// SIMATIC STEP 7 (V5.x) project PRACTICA PRESELECCIO
// CPU: CPU313 C-2 DP(1)
// station: P_ADR_BUS
// station: Hardware
// station: Equipo SIMATIC 300
// program: Programa S7(1)

SYMBOL_TABLE
"FLANCOS"	DB 1	DB 1
"P PRESELECCION"	I 0.0	BOOL
"EJECUTAR"	I 0.1	BOOL
"P EMERGENCIA"	I 0.2	BOOL
"Cycle Execution"	OB 1	OB 1
"SELECCION BOMBA 1"	Q 0.0	BOOL
"SELECCION BOMBA 2"	Q 0.1	BOOL
"SELECCION BOMBA 3"	Q 0.2	BOOL
"SELECCION BOMBA 4"	Q 0.3	BOOL
"EJECUCION BOMBA 1"	Q 0.4	BOOL
"EJECUCION BOMBA 2"	Q 0.5	BOOL
"EJECUCION BOMBA 3"	Q 0.6	BOOL
"EJECUCION BOMBA 4"	Q 0.7	BOOL
END_SYMBOL_TABLE

DATA_BLOCK "FLANCOS"	// DB 1
VERSION : 0.1
  STRUCT
   M0 : BOOL ;
   M1 : BOOL ;
   M2 : BOOL ;
   M3 : BOOL ;
   M4 : BOOL ;
   M5 : BOOL ;
   M6 : BOOL ;
   M7 : BOOL ;
   M10 : BOOL ;
   M11 : BOOL ;
   M12 : BOOL ;
   M13 : BOOL ;
   M14 : BOOL ;
   M15 : BOOL ;
   M16 : BOOL ;
   M17 : BOOL ;
   M20 : BOOL ;
   M21 : BOOL ;
   M22 : BOOL ;
   M23 : BOOL ;
   M24 : BOOL ;
   M25 : BOOL ;
   M26 : BOOL ;
   M27 : BOOL ;
  END_STRUCT ;	
BEGIN
END_DATA_BLOCK

ORGANIZATION_BLOCK "Cycle Execution"	// OB 1
TITLE = "Main Program Sweep (Cycle)"
VERSION : 0.1
VAR_TEMP
  OB1_EV_CLASS : BYTE ;	//Bits 0-3 = 1 (Coming event), Bits 4-7 = 1 (Event class 1)
  OB1_SCAN_1 : BYTE ;	//1 (Cold restart scan 1 of OB 1), 3 (Scan 2-n of OB 1)
  OB1_PRIORITY : BYTE ;	//Priority of OB Execution
  OB1_OB_NUMBR : BYTE ;	//1 (Organization block 1, OB1)
  OB1_RESERVED_1 : BYTE ;	//Reserved for system
  OB1_RESERVED_2 : BYTE ;	//Reserved for system
  OB1_PREV_CYCLE : INT ;	//Cycle time of previous OB1 scan (milliseconds)
  OB1_MIN_CYCLE : INT ;	//Minimum cycle time of OB1 (milliseconds)
  OB1_MAX_CYCLE : INT ;	//Maximum cycle time of OB1 (milliseconds)
  OB1_DATE_TIME : DATE_AND_TIME ;	//Date and time OB1 started
END_VAR
BEGIN
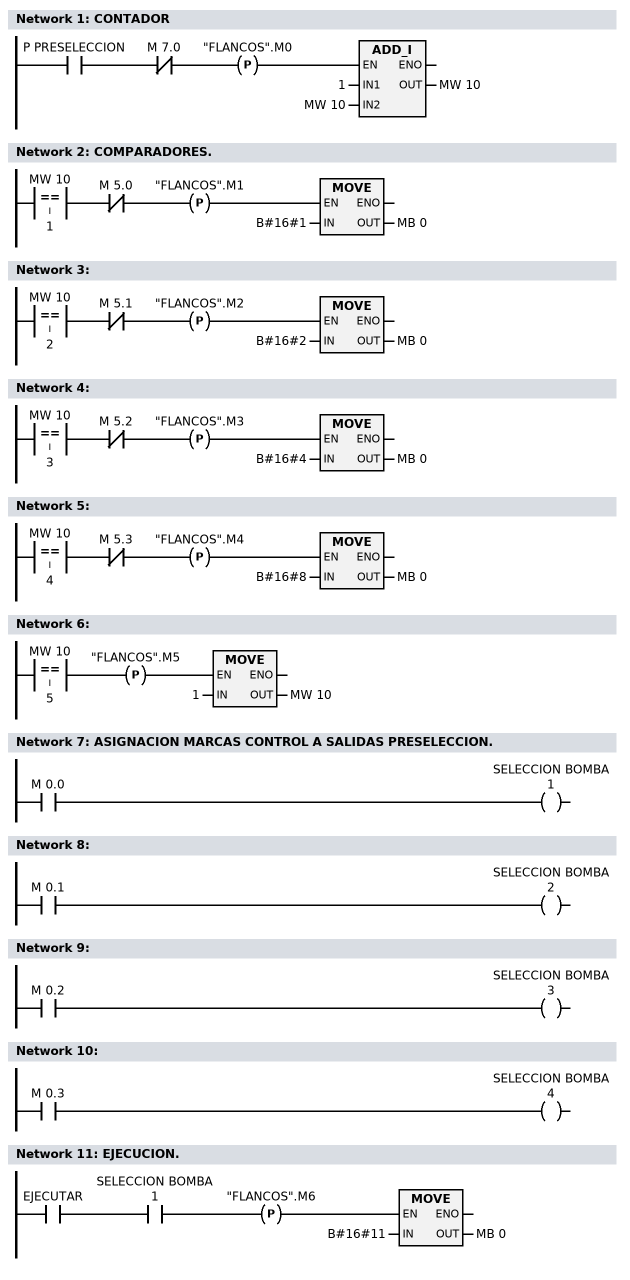
NETWORK
TITLE = CONTADOR
      A     "P PRESELECCION";
      AN    M 7.0;
      FP    "FLANCOS".M0;
      JNB   _001;
      L     1;
      L     MW 10;
      +I;
      T     MW 10;
_001: NOP   0;
NETWORK
TITLE = COMPARADORES.
      A(;
      L     MW 10;
      L     1;
      ==I;
      );
      AN    M 5.0;
      FP    "FLANCOS".M1;
      JNB   _002;
      L     B#16#1;
      T     MB 0;
_002: NOP   0;
NETWORK
TITLE =
      A(;
      L     MW 10;
      L     2;
      ==I;
      );
      AN    M 5.1;
      FP    "FLANCOS".M2;
      JNB   _003;
      L     B#16#2;
      T     MB 0;
_003: NOP   0;
NETWORK
TITLE =
      A(;
      L     MW 10;
      L     3;
      ==I;
      );
      AN    M 5.2;
      FP    "FLANCOS".M3;
      JNB   _004;
      L     B#16#4;
      T     MB 0;
_004: NOP   0;
NETWORK
TITLE =
      A(;
      L     MW 10;
      L     4;
      ==I;
      );
      AN    M 5.3;
      FP    "FLANCOS".M4;
      JNB   _005;
      L     B#16#8;
      T     MB 0;
_005: NOP   0;
NETWORK
TITLE =
      A(;
      L     MW 10;
      L     5;
      ==I;
      );
      FP    "FLANCOS".M5;
      JNB   _006;
      L     1;
      T     MW 10;
_006: NOP   0;
NETWORK
TITLE = ASIGNACION MARCAS CONTROL A SALIDAS PRESELECCION.
      A     M 0.0;
      =     "SELECCION BOMBA 1";
NETWORK
TITLE =
      A     M 0.1;
      =     "SELECCION BOMBA 2";
NETWORK
TITLE =
      A     M 0.2;
      =     "SELECCION BOMBA 3";
NETWORK
TITLE =
      A     M 0.3;
      =     "SELECCION BOMBA 4";
NETWORK
TITLE = EJECUCION.
      A     "EJECUTAR";
      A     "SELECCION BOMBA 1";
      FP    "FLANCOS".M6;
      JNB   _007;
      L     B#16#11;
      T     MB 0;
_007: NOP   0;
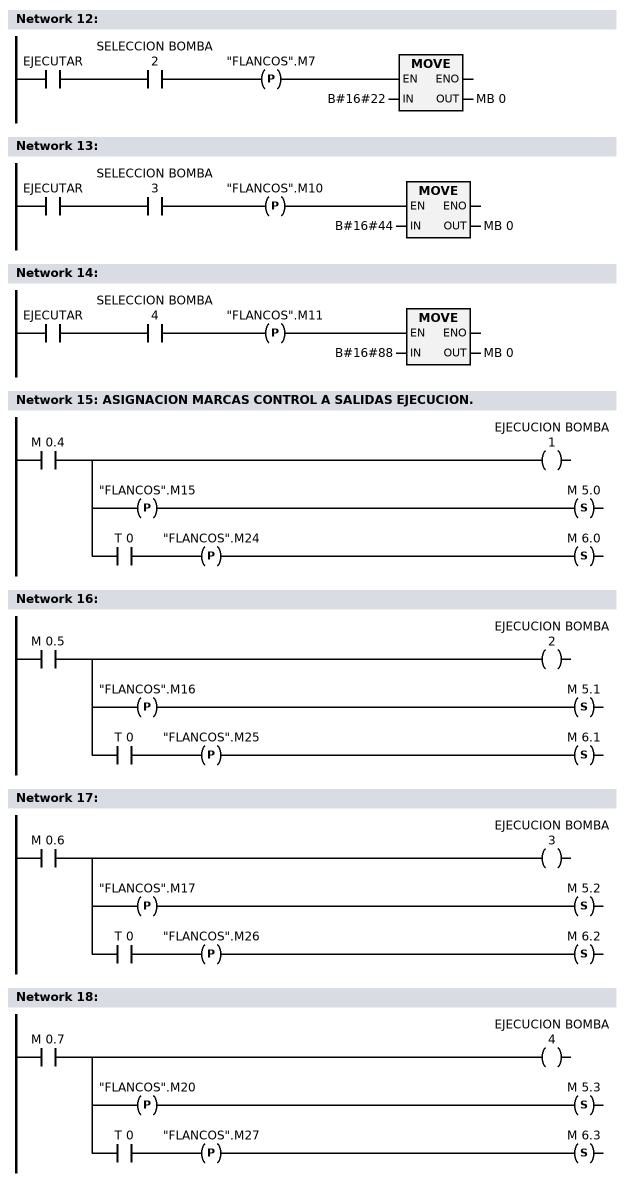
NETWORK
TITLE =
      A     "EJECUTAR";
      A     "SELECCION BOMBA 2";
      FP    "FLANCOS".M7;
      JNB   _008;
      L     B#16#22;
      T     MB 0;
_008: NOP   0;
NETWORK
TITLE =
      A     "EJECUTAR";
      A     "SELECCION BOMBA 3";
      FP    "FLANCOS".M10;
      JNB   _009;
      L     B#16#44;
      T     MB 0;
_009: NOP   0;
NETWORK
TITLE =
      A     "EJECUTAR";
      A     "SELECCION BOMBA 4";
      FP    "FLANCOS".M11;
      JNB   _00a;
      L     B#16#88;
      T     MB 0;
_00a: NOP   0;
NETWORK
TITLE = ASIGNACION MARCAS CONTROL A SALIDAS EJECUCION.
      A     M 0.4;
      =     L 20.0;
      A     L 20.0;
      BLD   102;
      =     "EJECUCION BOMBA 1";
      A     L 20.0;
      FP    "FLANCOS".M15;
      S     M 5.0;
      A     L 20.0;
      A     T 0;
      FP    "FLANCOS".M24;
      S     M 6.0;
NETWORK
TITLE =
      A     M 0.5;
      =     L 20.0;
      A     L 20.0;
      BLD   102;
      =     "EJECUCION BOMBA 2";
      A     L 20.0;
      FP    "FLANCOS".M16;
      S     M 5.1;
      A     L 20.0;
      A     T 0;
      FP    "FLANCOS".M25;
      S     M 6.1;
NETWORK
TITLE =
      A     M 0.6;
      =     L 20.0;
      A     L 20.0;
      BLD   102;
      =     "EJECUCION BOMBA 3";
      A     L 20.0;
      FP    "FLANCOS".M17;
      S     M 5.2;
      A     L 20.0;
      A     T 0;
      FP    "FLANCOS".M26;
      S     M 6.2;
NETWORK
TITLE =
      A     M 0.7;
      =     L 20.0;
      A     L 20.0;
      BLD   102;
      =     "EJECUCION BOMBA 4";
      A     L 20.0;
      FP    "FLANCOS".M20;
      S     M 5.3;
      A     L 20.0;
      A     T 0;
      FP    "FLANCOS".M27;
      S     M 6.3;
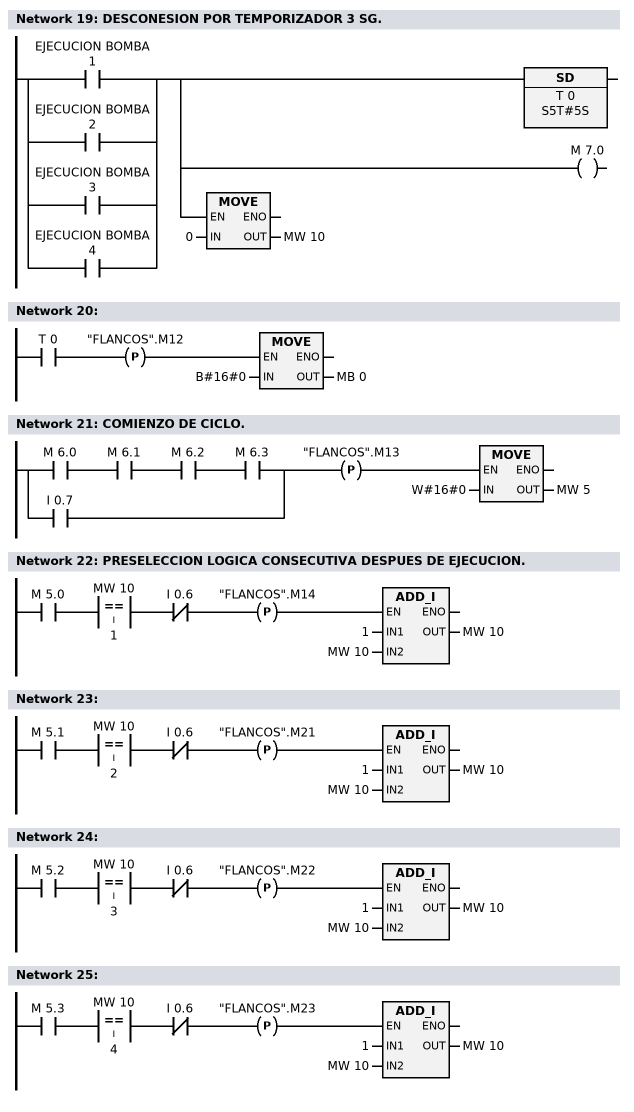
NETWORK
TITLE = DESCONESION POR TEMPORIZADOR 3 SG.
      O     "EJECUCION BOMBA 1";
      O     "EJECUCION BOMBA 2";
      O     "EJECUCION BOMBA 3";
      O     "EJECUCION BOMBA 4";
      =     L 20.0;
      A     L 20.0;
      BLD   102;
      L     S5T#5S;
      SD    T 0;
      A     L 20.0;
      BLD   102;
      =     M 7.0;
      A     L 20.0;
      JNB   _013;
      L     0;
      T     MW 10;
_013: NOP   0;
NETWORK
TITLE =
      A     T 0;
      FP    "FLANCOS".M12;
      JNB   _014;
      L     B#16#0;
      T     MB 0;
_014: NOP   0;
NETWORK
TITLE = COMIENZO DE CICLO.
      A(;
      A     M 6.0;
      A     M 6.1;
      A     M 6.2;
      A     M 6.3;
      O     I 0.7;
      );
      FP    "FLANCOS".M13;
      JNB   _015;
      L     W#16#0;
      T     MW 5;
_015: NOP   0;
NETWORK
TITLE = PRESELECCION LOGICA CONSECUTIVA DESPUES DE EJECUCION.
      A     M 5.0;
      A(;
      L     MW 10;
      L     1;
      ==I;
      );
      AN    I 0.6;
      FP    "FLANCOS".M14;
      JNB   _016;
      L     1;
      L     MW 10;
      +I;
      T     MW 10;
_016: NOP   0;
NETWORK
TITLE =
      A     M 5.1;
      A(;
      L     MW 10;
      L     2;
      ==I;
      );
      AN    I 0.6;
      FP    "FLANCOS".M21;
      JNB   _017;
      L     1;
      L     MW 10;
      +I;
      T     MW 10;
_017: NOP   0;
NETWORK
TITLE =
      A     M 5.2;
      A(;
      L     MW 10;
      L     3;
      ==I;
      );
      AN    I 0.6;
      FP    "FLANCOS".M22;
      JNB   _018;
      L     1;
      L     MW 10;
      +I;
      T     MW 10;
_018: NOP   0;
NETWORK
TITLE =
      A     M 5.3;
      A(;
      L     MW 10;
      L     4;
      ==I;
      );
      AN    I 0.6;
      FP    "FLANCOS".M23;
      JNB   _019;
      L     1;
      L     MW 10;
      +I;
      T     MW 10;
_019: NOP   0;
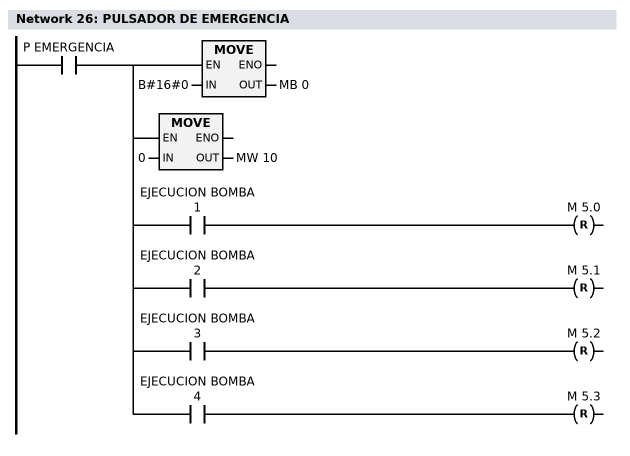
NETWORK
TITLE = PULSADOR DE EMERGENCIA
      A     "P EMERGENCIA";
      =     L 20.0;
      A     L 20.0;
      JNB   _01a;
      L     B#16#0;
      T     MB 0;
_01a: NOP   0;
      A     L 20.0;
      JNB   _01b;
      L     0;
      T     MW 10;
_01b: NOP   0;
      A     L 20.0;
      A     "EJECUCION BOMBA 1";
      R     M 5.0;
      A     L 20.0;
      A     "EJECUCION BOMBA 2";
      R     M 5.1;
      A     L 20.0;
      A     "EJECUCION BOMBA 3";
      R     M 5.2;
      A     L 20.0;
      A     "EJECUCION BOMBA 4";
      R     M 5.3;
END_ORGANIZATION_BLOCK
